SYSTEM TankControlDemo
  (* Version 1.0, Author, 4DIAC-Consortium *)
  APPLICATION TankControl
    FBS
      F_NOT_1_1 : F_NOT;
      FB_CTRL_PID_1_1 : FB_CTRL_PID(SUP := 0.1, OFS := 0, KP := 2, TN := 1, TV := 0.02, LIM_L := 0.0, LIM_H := 100.0);
      CNV_VALVEPOS_1 : FB_REAL_UINT;
      VALVE_VIEW_1 : VALVE_VIEW(DIA := 50, FGD := [0,255,0]);
      TANK_VIEW_1 : MECH_VIEW(STYLE := VSTYLE#CYLINDER, WKPC := [0,0,255], BKGD := [255,255,255], LEN := 2, DIR := 3);
      TANK_SIM_MDL_1 : TANK_MDL(DT := t#250ms, TF := T#1s);
      CNV_LEVEL_1 : FB_REAL_UINT;
      SUB_VALVE_MODE_1 : SUBSCRIBE_1(QI := TRUE, ID := sfp[feed_valve_control.mode]);
      SUB_LEVEL_SETPOINT_1 : SUBSCRIBE_1(QI := TRUE, ID := sfp[level.set_point]);
      SUB_VALVE_MANUALPOS_1 : SUBSCRIBE_1(QI := TRUE, ID := sfp[feed_valve_control.manual_set_position]);
      CNV_VALVE_MODE_1 : BOOL2BOOL;
      SUB_PUMP_SETSPEED_1 : SUBSCRIBE_1(QI := TRUE, ID := sfp[pump.set_speed]);
      CNV_PUMP_SETSPEED_1 : F_LREAL_TO_UINT;
      PUB_VALVE_SETPOS_1 : PUBLISH_1(QI := TRUE, ID := sfp[feed_valve_control.set_position]);
      CNV_LEVEL_MEASURED_1 : F_REAL_TO_LREAL;
      PUB_LEVEL_MEASURED_1 : PUBLISH_1(QI := TRUE, ID := sfp[level.measured]);
      SCALE_PUMP_SETSPEED_1 : UNSCALE(MAX := 360);
      SHAFT_MDL_1 : SHAFT_MDL(DT := T#100ms);
      XSPACE_1 : XSPACE(DIMS := [3,1], DIA := 20);
      PIPE_VIEW_1 : PIPE_VIEW(DIR := [0,1]);
      PUMP_DEV_VIEW_1 : PUMP_VIEW(FGD := [255,0,0], IX := [0,0,255]);
    END_FBS
    EVENT_CONNECTIONS
      VALVE_VIEW_1.CNF TO TANK_VIEW_1.REQ;
      VALVE_VIEW_1.INITO TO TANK_VIEW_1.INIT;
      TANK_SIM_MDL_1.EO TO FB_CTRL_PID_1_1.REQ;
      CNV_LEVEL_1.CNF TO CNV_VALVEPOS_1.REQ;
      CNV_LEVEL_MEASURED_1.CNF TO PUB_LEVEL_MEASURED_1.REQ;
      F_NOT_1_1.CNF TO FB_CTRL_PID_1_1.RST;
      CNV_VALVEPOS_1.CNF TO VALVE_VIEW_1.REQ;
      SUB_VALVE_MODE_1.IND TO CNV_VALVE_MODE_1.REQ;
      SUB_PUMP_SETSPEED_1.IND TO CNV_PUMP_SETSPEED_1.REQ;
      TANK_VIEW_1.INITO TO TANK_SIM_MDL_1.START;
      TANK_SIM_MDL_1.EO TO CNV_LEVEL_1.REQ;
      SUB_LEVEL_SETPOINT_1.IND TO FB_CTRL_PID_1_1.RST;
      SUB_VALVE_MANUALPOS_1.IND TO FB_CTRL_PID_1_1.RST;
      CNV_VALVE_MODE_1.CNF TO F_NOT_1_1.REQ;
      FB_CTRL_PID_1_1.CNF TO PUB_VALVE_SETPOS_1.REQ;
      TANK_SIM_MDL_1.EO TO CNV_LEVEL_MEASURED_1.REQ;
      CNV_PUMP_SETSPEED_1.CNF TO SCALE_PUMP_SETSPEED_1.REQ;
      PUB_VALVE_SETPOS_1.INITO TO PUB_LEVEL_MEASURED_1.INIT;
      PUB_LEVEL_MEASURED_1.INITO TO SUB_LEVEL_SETPOINT_1.INIT;
      SUB_LEVEL_SETPOINT_1.INITO TO SUB_VALVE_MANUALPOS_1.INIT;
      SUB_VALVE_MANUALPOS_1.INITO TO SUB_VALVE_MODE_1.INIT;
      SUB_VALVE_MODE_1.INITO TO SUB_PUMP_SETSPEED_1.INIT;
      SUB_LOCAL_ACTLEVEL.IND TO CNV_LEVEL_MEASURED_1.REQ;
      CNV_PUMP_SETSPEED_1.CNF TO PUB_LOCAL_PUMPSPEED.REQ;
      START.COLD TO PUB_VALVE_SETPOS_1.INIT;
      START.WARM TO PUB_VALVE_SETPOS_1.INIT;
      SUBSCRIBE_1_6.INITO TO XSPACE_1.INIT;
      SUBSCRIBE_1_6.IND TO SCALE_PUMP_SETSPEED_1.REQ;
      XSPACE_1.INITO TO PIPE_VIEW_1.INIT;
      PIPE_VIEW_1.INITO TO PUMP_DEV_VIEW_1.INIT;
      SHAFT_MDL_1.EO TO PUMP_DEV_VIEW_1.REQ;
      PUMP_DEV_VIEW_1.INITO TO SHAFT_MDL_1.START;
    END_CONNECTIONS
    DATA_CONNECTIONS
      CNV_LEVEL_1.OUT TO TANK_VIEW_1.POS;
      SUB_VALVE_MODE_1.RD_1 TO CNV_VALVE_MODE_1.IN;
      F_NOT_1_1.OUT TO FB_CTRL_PID_1_1.MAN;
      CNV_LEVEL_MEASURED_1.OUT TO PUB_LEVEL_MEASURED_1.SD_1;
      TANK_SIM_MDL_1.LEVEL TO FB_CTRL_PID_1_1.ACT;
      CNV_VALVEPOS_1.OUT TO VALVE_VIEW_1.POS;
      SUB_PUMP_SETSPEED_1.RD_1 TO CNV_PUMP_SETSPEED_1.IN;
      TANK_SIM_MDL_1.LEVEL TO CNV_LEVEL_1.IN;
      FB_CTRL_PID_1_1.Y TO TANK_SIM_MDL_1.FEED;
      FB_CTRL_PID_1_1.Y TO CNV_VALVEPOS_1.IN;
      SUB_LEVEL_SETPOINT_1.RD_1 TO FB_CTRL_PID_1_1.SET;
      SUB_VALVE_MANUALPOS_1.RD_1 TO FB_CTRL_PID_1_1.M_I;
      CNV_VALVE_MODE_1.OUT TO F_NOT_1_1.IN;
      FB_CTRL_PID_1_1.Y TO PUB_VALVE_SETPOS_1.SD_1;
      TANK_SIM_MDL_1.LEVEL TO CNV_LEVEL_MEASURED_1.IN;
      CNV_PUMP_SETSPEED_1.OUT TO TANK_SIM_MDL_1.DRAW;
      CNV_PUMP_SETSPEED_1.OUT TO SCALE_PUMP_SETSPEED_1.IN;
      SUB_LOCAL_ACTLEVEL.RD_1 TO CNV_LEVEL_MEASURED_1.IN;
      CNV_PUMP_SETSPEED_1.OUT TO PUB_LOCAL_PUMPSPEED.SD_1;
      SUBSCRIBE_1_6.RD_1 TO SCALE_PUMP_SETSPEED_1.IN;
      SCALE_PUMP_SETSPEED_1.OUT TO SHAFT_MDL_1.V;
      SHAFT_MDL_1.POS TO PUMP_DEV_VIEW_1.ANGLE;
    END_CONNECTIONS
  END_APPLICATION
  DEVICE TankSimulation : RMT_FRAME(BOUNDS := [315,100,175,260], MGR_ID := "localhost:61500")
    {SET_ATTRIBUTE(Profile, HOLOBLOC)}
    RESOURCE TankValveSim : VIEW_PANEL(DIA := 75, SIZE := [3,2])
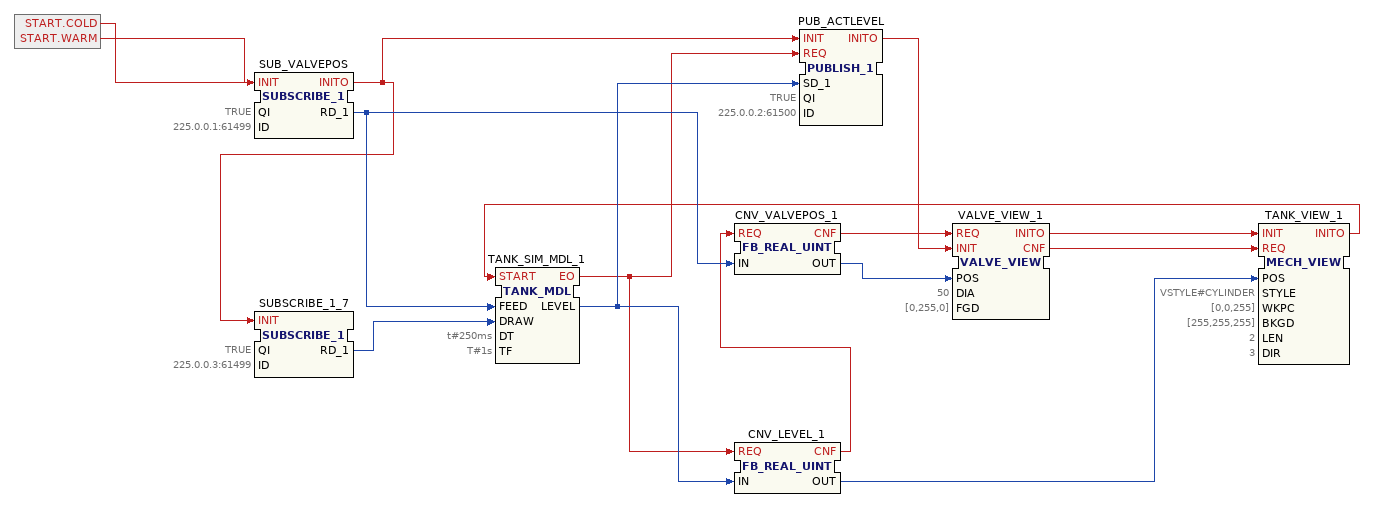
      FBS
        PUB_ACTLEVEL : PUBLISH_1(QI := TRUE, ID := 225.0.0.2:61500);
        SUB_VALVEPOS : SUBSCRIBE_1(QI := TRUE, ID := 225.0.0.1:61499);
        SUBSCRIBE_1_7 : SUBSCRIBE_1(QI := TRUE, ID := 225.0.0.3:61499);
        TANK_SIM_MDL_1 : TANK_MDL(DT := t#250ms, TF := T#1s);
        CNV_LEVEL_1 : FB_REAL_UINT;
        CNV_VALVEPOS_1 : FB_REAL_UINT;
        VALVE_VIEW_1 : VALVE_VIEW(DIA := 50, FGD := [0,255,0]);
        TANK_VIEW_1 : MECH_VIEW(STYLE := VSTYLE#CYLINDER, WKPC := [0,0,255], BKGD := [255,255,255], LEN := 2, DIR := 3);
      END_FBS
      EVENT_CONNECTIONS
        START.COLD TO SUB_VALVEPOS.INIT;
        START.WARM TO SUB_VALVEPOS.INIT;
        SUB_VALVEPOS.INITO TO PUB_ACTLEVEL.INIT;
        SUB_VALVEPOS.INITO TO SUBSCRIBE_1_7.INIT;
        TANK_SIM_MDL_1.EO TO CNV_LEVEL_1.REQ;
        CNV_LEVEL_1.CNF TO CNV_VALVEPOS_1.REQ;
        CNV_VALVEPOS_1.CNF TO VALVE_VIEW_1.REQ;
        VALVE_VIEW_1.INITO TO TANK_VIEW_1.INIT;
        VALVE_VIEW_1.CNF TO TANK_VIEW_1.REQ;
        TANK_VIEW_1.INITO TO TANK_SIM_MDL_1.START;
        PUB_ACTLEVEL.INITO TO VALVE_VIEW_1.INIT;
        TANK_SIM_MDL_1.EO TO PUB_ACTLEVEL.REQ;
      END_CONNECTIONS
      DATA_CONNECTIONS
        TANK_SIM_MDL_1.LEVEL TO CNV_LEVEL_1.IN;
        CNV_VALVEPOS_1.OUT TO VALVE_VIEW_1.POS;
        CNV_LEVEL_1.OUT TO TANK_VIEW_1.POS;
        TANK_SIM_MDL_1.LEVEL TO PUB_ACTLEVEL.SD_1;
        SUB_VALVEPOS.RD_1 TO CNV_VALVEPOS_1.IN;
        SUB_VALVEPOS.RD_1 TO TANK_SIM_MDL_1.FEED;
        SUBSCRIBE_1_7.RD_1 TO TANK_SIM_MDL_1.DRAW;
      END_CONNECTIONS
    END_RESOURCE
    RESOURCE PumpSim : VIEW_PANEL(DIA := 50, SIZE := [4,1])
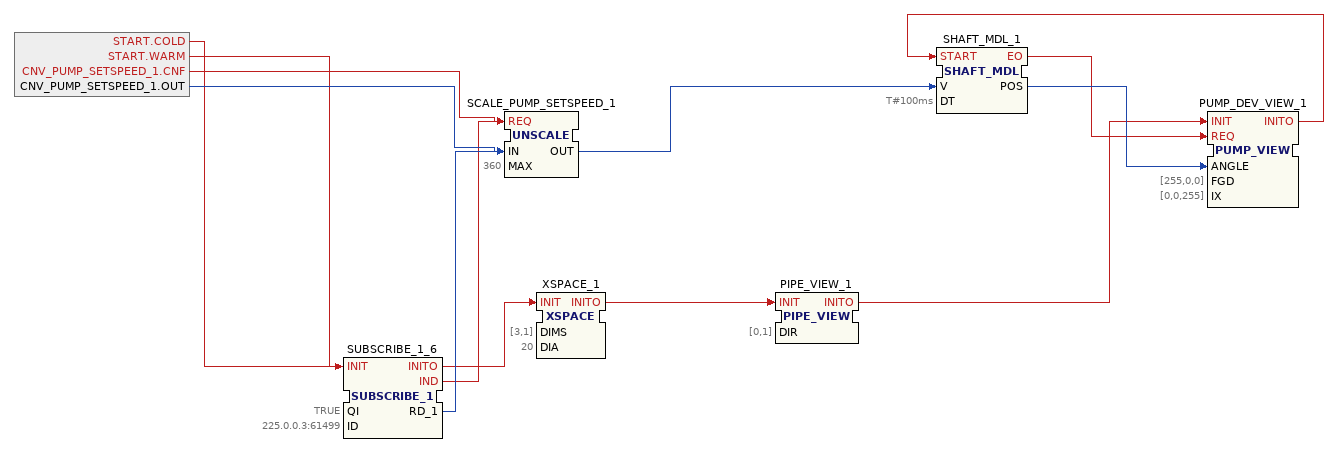
      FBS
        SUBSCRIBE_1_6 : SUBSCRIBE_1(QI := TRUE, ID := 225.0.0.3:61499);
        SCALE_PUMP_SETSPEED_1 : UNSCALE(MAX := 360);
        SHAFT_MDL_1 : SHAFT_MDL(DT := T#100ms);
        XSPACE_1 : XSPACE(DIMS := [3,1], DIA := 20);
        PIPE_VIEW_1 : PIPE_VIEW(DIR := [0,1]);
        PUMP_DEV_VIEW_1 : PUMP_VIEW(FGD := [255,0,0], IX := [0,0,255]);
      END_FBS
      EVENT_CONNECTIONS
        START.COLD TO SUBSCRIBE_1_6.INIT;
        START.WARM TO SUBSCRIBE_1_6.INIT;
        SUBSCRIBE_1_6.INITO TO XSPACE_1.INIT;
        SUBSCRIBE_1_6.IND TO SCALE_PUMP_SETSPEED_1.REQ;
        CNV_PUMP_SETSPEED_1.CNF TO SCALE_PUMP_SETSPEED_1.REQ;
        XSPACE_1.INITO TO PIPE_VIEW_1.INIT;
        PIPE_VIEW_1.INITO TO PUMP_DEV_VIEW_1.INIT;
        SHAFT_MDL_1.EO TO PUMP_DEV_VIEW_1.REQ;
        PUMP_DEV_VIEW_1.INITO TO SHAFT_MDL_1.START;
      END_CONNECTIONS
      DATA_CONNECTIONS
        SUBSCRIBE_1_6.RD_1 TO SCALE_PUMP_SETSPEED_1.IN;
        CNV_PUMP_SETSPEED_1.OUT TO SCALE_PUMP_SETSPEED_1.IN;
        SCALE_PUMP_SETSPEED_1.OUT TO SHAFT_MDL_1.V;
        SHAFT_MDL_1.POS TO PUMP_DEV_VIEW_1.ANGLE;
      END_CONNECTIONS
    END_RESOURCE
  END_DEVICE
  DEVICE Controller_1 : RMT_DEV(MGR_ID := "localhost:61499")
    {SET_ATTRIBUTE(Profile, HOLOBLOC)}
    RESOURCE PID : EMB_RES
      FBS
        SUB_LOCAL_ACTLEVEL : SUBSCRIBE_1(QI := TRUE, ID := 225.0.0.2:61500);
        PUB_LOCAL_VALVEPOS_IN : PUBLISH_1(QI := TRUE, ID := 225.0.0.1:61499);
        PUB_LOCAL_PUMPSPEED : PUBLISH_1(QI := TRUE, ID := 225.0.0.3:61499);
        SUB_VALVE_MODE_1 : SUBSCRIBE_1(QI := TRUE, ID := sfp[feed_valve_control.mode]);
        SUB_LEVEL_SETPOINT_1 : SUBSCRIBE_1(QI := TRUE, ID := sfp[level.set_point]);
        SUB_VALVE_MANUALPOS_1 : SUBSCRIBE_1(QI := TRUE, ID := sfp[feed_valve_control.manual_set_position]);
        CNV_VALVE_MODE_1 : BOOL2BOOL;
        SUB_PUMP_SETSPEED_1 : SUBSCRIBE_1(QI := TRUE, ID := sfp[pump.set_speed]);
        CNV_PUMP_SETSPEED_1 : F_LREAL_TO_UINT;
        PUB_VALVE_SETPOS_1 : PUBLISH_1(QI := TRUE, ID := sfp[feed_valve_control.set_position]);
        CNV_LEVEL_MEASURED_1 : F_REAL_TO_LREAL;
        PUB_LEVEL_MEASURED_1 : PUBLISH_1(QI := TRUE, ID := sfp[level.measured]);
        FB_CTRL_PID_1_1 : FB_CTRL_PID(SUP := 0.1, OFS := 0, KP := 2, TN := 1, TV := 0.02, LIM_L := 0.0, LIM_H := 100.0);
        F_NOT_1_1 : F_NOT;
      END_FBS
      EVENT_CONNECTIONS
        START.COLD TO SUB_LOCAL_ACTLEVEL.INIT;
        START.WARM TO SUB_LOCAL_ACTLEVEL.INIT;
        SUB_LEVEL_SETPOINT_1.IND TO FB_CTRL_PID_1_1.RST;
        SUB_VALVE_MANUALPOS_1.IND TO FB_CTRL_PID_1_1.RST;
        FB_CTRL_PID_1_1.CNF TO PUB_VALVE_SETPOS_1.REQ;
        CNV_VALVE_MODE_1.CNF TO F_NOT_1_1.REQ;
        F_NOT_1_1.CNF TO FB_CTRL_PID_1_1.RST;
        SUB_LOCAL_ACTLEVEL.INITO TO PUB_LOCAL_PUMPSPEED.INIT;
        PUB_LOCAL_PUMPSPEED.INITO TO PUB_LOCAL_VALVEPOS_IN.INIT;
        SUB_LOCAL_ACTLEVEL.IND TO CNV_LEVEL_MEASURED_1.REQ;
        CNV_PUMP_SETSPEED_1.CNF TO PUB_LOCAL_PUMPSPEED.REQ;
        FB_CTRL_PID_1_1.CNF TO PUB_LOCAL_VALVEPOS_IN.REQ;
        START.COLD TO PUB_VALVE_SETPOS_1.INIT;
        START.WARM TO PUB_VALVE_SETPOS_1.INIT;
        START.COLD TO FB_CTRL_PID_1_1.INIT;
        START.WARM TO FB_CTRL_PID_1_1.INIT;
        SUB_LOCAL_ACTLEVEL.IND TO FB_CTRL_PID_1_1.REQ;
        TANK_SIM_MDL_1.EO TO CNV_LEVEL_MEASURED_1.REQ;
        CNV_PUMP_SETSPEED_1.CNF TO SCALE_PUMP_SETSPEED_1.REQ;
        PUB_VALVE_SETPOS_1.INITO TO PUB_LEVEL_MEASURED_1.INIT;
        PUB_LEVEL_MEASURED_1.INITO TO SUB_LEVEL_SETPOINT_1.INIT;
        SUB_LEVEL_SETPOINT_1.INITO TO SUB_VALVE_MANUALPOS_1.INIT;
        SUB_VALVE_MANUALPOS_1.INITO TO SUB_VALVE_MODE_1.INIT;
        SUB_VALVE_MODE_1.INITO TO SUB_PUMP_SETSPEED_1.INIT;
      END_CONNECTIONS
      DATA_CONNECTIONS
        SUB_LEVEL_SETPOINT_1.RD_1 TO FB_CTRL_PID_1_1.SET;
        SUB_VALVE_MANUALPOS_1.RD_1 TO FB_CTRL_PID_1_1.M_I;
        FB_CTRL_PID_1_1.Y TO PUB_VALVE_SETPOS_1.SD_1;
        CNV_VALVE_MODE_1.OUT TO F_NOT_1_1.IN;
        F_NOT_1_1.OUT TO FB_CTRL_PID_1_1.MAN;
        SUB_LOCAL_ACTLEVEL.RD_1 TO CNV_LEVEL_MEASURED_1.IN;
        SUB_LOCAL_ACTLEVEL.RD_1 TO FB_CTRL_PID_1_1.ACT;
        CNV_PUMP_SETSPEED_1.OUT TO PUB_LOCAL_PUMPSPEED.SD_1;
        FB_CTRL_PID_1_1.Y TO PUB_LOCAL_VALVEPOS_IN.SD_1;
        TANK_SIM_MDL_1.LEVEL TO CNV_LEVEL_MEASURED_1.IN;
        CNV_PUMP_SETSPEED_1.OUT TO TANK_SIM_MDL_1.DRAW;
        CNV_PUMP_SETSPEED_1.OUT TO SCALE_PUMP_SETSPEED_1.IN;
      END_CONNECTIONS
    END_RESOURCE
  END_DEVICE
  MAPPINGS
    TankControl.F_NOT_1_1 ON Controller_1.PID.F_NOT_1_1;
    TankControl.FB_CTRL_PID_1_1 ON Controller_1.PID.FB_CTRL_PID_1_1;
    TankControl.CNV_VALVEPOS_1 ON TankSimulation.TankValveSim.CNV_VALVEPOS_1;
    TankControl.VALVE_VIEW_1 ON TankSimulation.TankValveSim.VALVE_VIEW_1;
    TankControl.TANK_VIEW_1 ON TankSimulation.TankValveSim.TANK_VIEW_1;
    TankControl.TANK_SIM_MDL_1 ON TankSimulation.TankValveSim.TANK_SIM_MDL_1;
    TankControl.CNV_LEVEL_1 ON TankSimulation.TankValveSim.CNV_LEVEL_1;
  END_MAPPINGS
  SEGMENTS
    Ethernet : Ethernet;
  END_SEGMENTS
  LINKS
    Controller_1 => Ethernet;
    TankSimulation => Ethernet;
  END_LINKS
END_SYSTEM
